PROGRAM PRG_SENSORS
VAR
        // Sensor Range in Psi
    CDA_SENS_PRESS_RANGE : REAL := 200;
    NITR_SENS_PRESS_RANGE: REAL := 200;
    H2O_SENS_PRESS_RANGE: REAL := 200;

    // Mim pressure setpoint in Psi
    CDA_SENS_MIN_PRESS_SP: REAL := 30;
    NITR_SENS_MIN_PRESS_SP: REAL := 15;
    H2O_SENS_MIN_PRESS_SP: REAL := 15;

    // Maximum pressure setpoint in Psi
    CDA_SENS_MAX_PRESS_SP: REAL := 160;
    NITR_SENS_MAX_PRESS_SP: REAL := 55;
    H2O_SENS_MAX_PRESS_SP: REAL := 80;

    // Press default setpoint in Psi
    CDA_SENS_DEFAULT_SP: REAL := 60;
    NITR_SENS_DEFAULT_SP: REAL := 25;
    H2O_SENS_DEFAULT_SP: REAL := 30;


END_VAR


GEM1_AIR_1(rDefaultSP:= CDA_SENS_DEFAULT_SP);
GEM1_AIR_2(rDefaultSP:= CDA_SENS_DEFAULT_SP);

GEM2_N2_1 (rDefaultSP:= NITR_SENS_DEFAULT_SP);
GEM2_N2_2 (rDefaultSP:= NITR_SENS_DEFAULT_SP);

END_PROGRAM

(* stored: Version 1.1.0.1, ProductVersion 3.1.4022.16
   POU PRG_SENSORS: Id {06b92b62-a281-4dd8-802c-ea3d5a53b2c1}, SpecialFunc None *)
